// TIA Portal V20 export
DATA_BLOCK "ET500SP_508"   // DB230
// stored: MemoryReserve 100
   VAR
      "SP508.00 PHMI-1 EMERGENCY STOP" : Bool;
      "SP508.01 PHMI-1 ENABLE SWITCH" : Bool;
      "SP508.02 PHMI-2 EMERGENCY STOP" : Bool;
      "SP508.03 PHMI-2 ENABLE SWITCH" : Bool;
      SPARE1 : Bool;
      SPARE2 : Bool;
      SPARE3 : Bool;
      SPARE4 : Bool;
   END_VAR
BEGIN
END_DATA_BLOCK
